Universal Robots PolyScope program: production_mix.urp

Program production_mix (installation=default directory=/home/ur/ursim-current/programs createdIn=5.16.1 lastSavedIn=5.16.1 robotSerialNumber=20195299999)
Calibrated DH parameters: a=[0, -0.6127, -0.57155, 0, 0, 0]; d=[0.1807, 0, 0, 0.17415, 0.11985, 0.11655]; alpha=[1.570796, 0, 0, 1.570796, -1.570796, 0]; deltaTheta=[0, 0, 0, 0, 0, 0]
InitVariablesNode
Robot Program (runOnlyOnce=false)
  Script file /home/ur/ursim-current/programs/production_tasks.script
    | square_count = 0
    | triangle_count = 0
    | circle_count = 0
    | square_target = 0
    | triangle_target = 0
    | circle_target = 0
    | 
    | def square_task():
    |     square_count = square_count + 1
    |     sleep(1)
    | end
    | 
    | def triangle_task():
    |     triangle_count = triangle_count + 1
    |     sleep(1)
    | end
    | 
    | def circle_task():
    |     circle_count = circle_count + 1
    |     sleep(1)
    | end
    | 
    | def start_task():
    |     while square_count < square_target or triangle_count < triangle_target or circle_count < circle_target:
    |     	if square_count < square_target:
    |             square_task()
    | 	    end
    | 
    | 	    if triangle_count < triangle_target:
    |             triangle_task()
    | 	    end
    | 
    | 	    if circle_count < circle_target:
    |             circle_task()
    | 	    end
    |     end
    | end
    | 
    | def reset_task():
    |     square_count = 0
    |     triangle_count = 0
    |     circle_count = 0
    |     square_target = 0
    |     triangle_target = 0
    |     circle_target = 0
    | end
  URCap HMI (Robpod HMI URcap, Robpod Cloud) dataModel(robpod.hmi.stop.main.loop=true, robpod.hmi.selected=/home/ur/ursim-current/programs/prduction_mix_hmi.hmi)
